PROGRAM MAIN
VAR_INPUT
	SysCommand			:SystemCommand;
	SkillCommand		:ObjectMode;
	testProcessValue	:Prozessvariablen; 
	
	Switch				:BOOL;
	
	
END_VAR

Anlage();
TestAblauf();

END_PROGRAM

(* stored: Version 1.1.0.1
   POU MAIN: Id {8cc3ee42-67a9-4667-b58e-96feb4991c55}, SpecialFunc None *)
